// SIMATIC S7-200 SMART project (STEP 7-Micro/WIN SMART), CPU CR40

SYMBOL_TABLE 系统符号
Always_On        SM0.0    // 始终接通
First_Scan_On    SM0.1    // 仅在第一个扫描周期时接通
END_SYMBOL_TABLE

ORGANIZATION_BLOCK MAIN:OB1
TITLE=程序注释
BEGIN
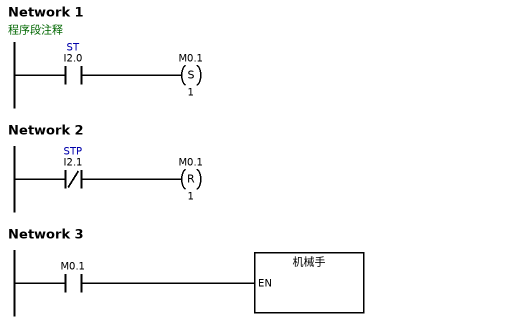
Network 1
// 程序段注释
LD     ST:I2.0
S      M0.1, 1
Network 2
LDN    STP:I2.1
R      M0.1, 1
Network 3
// (network saved uncompiled; LAD cells follow)
// row 0: c0 -| |- M0.1  c1 --  c2 [机械手 EN:=power@row0]
END_ORGANIZATION_BLOCK

SUBROUTINE_BLOCK 机械手:SBR0
TITLE=初始化，机械手复位
BEGIN
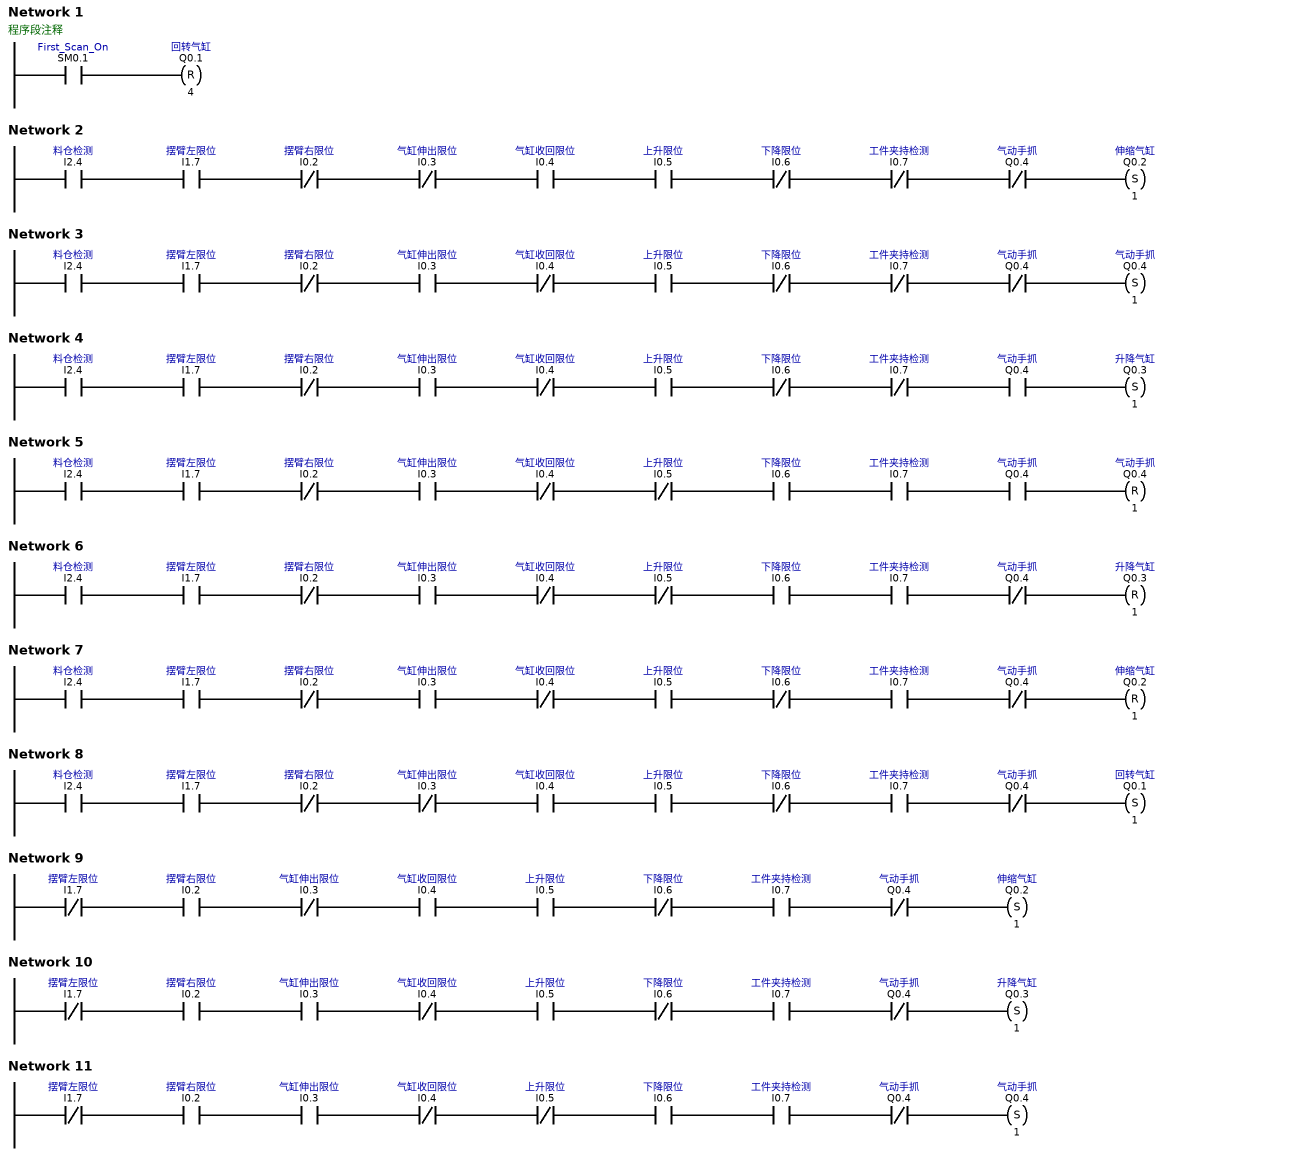
Network 1
// 程序段注释
LD     First_Scan_On:SM0.1
R      回转气缸:Q0.1, 4
Network 2
LD     料仓检测:I2.4
A      摆臂左限位:I1.7
AN     摆臂右限位:I0.2
AN     气缸伸出限位:I0.3
A      气缸收回限位:I0.4
A      上升限位:I0.5
AN     下降限位:I0.6
AN     工件夹持检测:I0.7
AN     气动手抓:Q0.4
S      伸缩气缸:Q0.2, 1
Network 3
LD     料仓检测:I2.4
A      摆臂左限位:I1.7
AN     摆臂右限位:I0.2
A      气缸伸出限位:I0.3
AN     气缸收回限位:I0.4
A      上升限位:I0.5
AN     下降限位:I0.6
AN     工件夹持检测:I0.7
AN     气动手抓:Q0.4
S      气动手抓:Q0.4, 1
Network 4
LD     料仓检测:I2.4
A      摆臂左限位:I1.7
AN     摆臂右限位:I0.2
A      气缸伸出限位:I0.3
AN     气缸收回限位:I0.4
A      上升限位:I0.5
AN     下降限位:I0.6
AN     工件夹持检测:I0.7
A      气动手抓:Q0.4
S      升降气缸:Q0.3, 1
Network 5
// 
// 
LD     料仓检测:I2.4
A      摆臂左限位:I1.7
AN     摆臂右限位:I0.2
A      气缸伸出限位:I0.3
AN     气缸收回限位:I0.4
AN     上升限位:I0.5
A      下降限位:I0.6
A      工件夹持检测:I0.7
A      气动手抓:Q0.4
R      气动手抓:Q0.4, 1
Network 6
// 
// 
LD     料仓检测:I2.4
A      摆臂左限位:I1.7
AN     摆臂右限位:I0.2
A      气缸伸出限位:I0.3
AN     气缸收回限位:I0.4
AN     上升限位:I0.5
A      下降限位:I0.6
A      工件夹持检测:I0.7
AN     气动手抓:Q0.4
R      升降气缸:Q0.3, 1
Network 7
// 
// 
LD     料仓检测:I2.4
A      摆臂左限位:I1.7
AN     摆臂右限位:I0.2
A      气缸伸出限位:I0.3
AN     气缸收回限位:I0.4
A      上升限位:I0.5
AN     下降限位:I0.6
A      工件夹持检测:I0.7
AN     气动手抓:Q0.4
R      伸缩气缸:Q0.2, 1
Network 8
// 
// 
LD     料仓检测:I2.4
A      摆臂左限位:I1.7
AN     摆臂右限位:I0.2
AN     气缸伸出限位:I0.3
A      气缸收回限位:I0.4
A      上升限位:I0.5
AN     下降限位:I0.6
A      工件夹持检测:I0.7
AN     气动手抓:Q0.4
S      回转气缸:Q0.1, 1
Network 9
// 
// 
// 
LDN    摆臂左限位:I1.7
A      摆臂右限位:I0.2
AN     气缸伸出限位:I0.3
A      气缸收回限位:I0.4
A      上升限位:I0.5
AN     下降限位:I0.6
A      工件夹持检测:I0.7
AN     气动手抓:Q0.4
S      伸缩气缸:Q0.2, 1
Network 10
// 
// 
// 
LDN    摆臂左限位:I1.7
A      摆臂右限位:I0.2
A      气缸伸出限位:I0.3
AN     气缸收回限位:I0.4
A      上升限位:I0.5
AN     下降限位:I0.6
A      工件夹持检测:I0.7
AN     气动手抓:Q0.4
S      升降气缸:Q0.3, 1
Network 11
// 
// 
// 
LDN    摆臂左限位:I1.7
A      摆臂右限位:I0.2
A      气缸伸出限位:I0.3
AN     气缸收回限位:I0.4
AN     上升限位:I0.5
A      下降限位:I0.6
A      工件夹持检测:I0.7
AN     气动手抓:Q0.4
S      气动手抓:Q0.4, 1
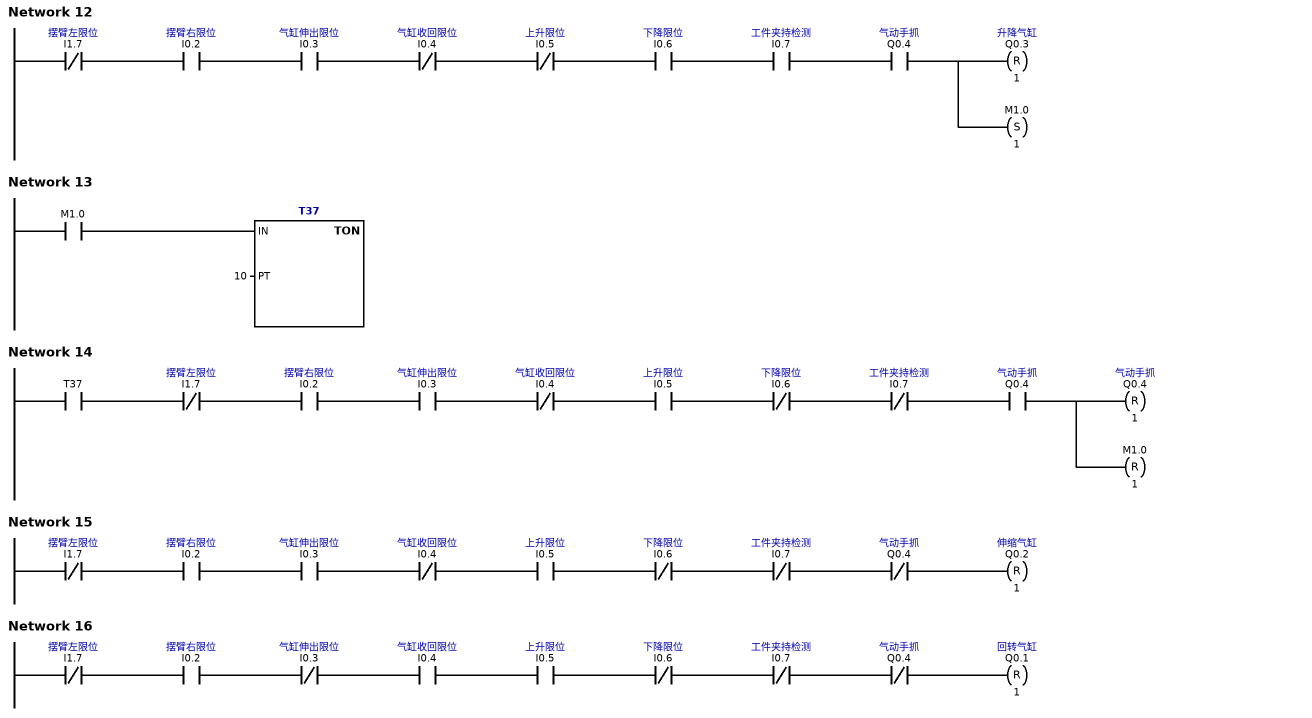
Network 12
// 
// 
// 
LDN    摆臂左限位:I1.7
A      摆臂右限位:I0.2
A      气缸伸出限位:I0.3
AN     气缸收回限位:I0.4
AN     上升限位:I0.5
A      下降限位:I0.6
A      工件夹持检测:I0.7
A      气动手抓:Q0.4
R      升降气缸:Q0.3, 1
S      M1.0, 1
Network 13
LD     M1.0
TON    T37, 10
Network 14
// 
// 
// 
LD     T37
AN     摆臂左限位:I1.7
A      摆臂右限位:I0.2
A      气缸伸出限位:I0.3
AN     气缸收回限位:I0.4
A      上升限位:I0.5
AN     下降限位:I0.6
AN     工件夹持检测:I0.7
A      气动手抓:Q0.4
R      气动手抓:Q0.4, 1
R      M1.0, 1
Network 15
// 
// 
// 
LDN    摆臂左限位:I1.7
A      摆臂右限位:I0.2
A      气缸伸出限位:I0.3
AN     气缸收回限位:I0.4
A      上升限位:I0.5
AN     下降限位:I0.6
AN     工件夹持检测:I0.7
AN     气动手抓:Q0.4
R      伸缩气缸:Q0.2, 1
Network 16
// 
// 
// 
LDN    摆臂左限位:I1.7
A      摆臂右限位:I0.2
AN     气缸伸出限位:I0.3
A      气缸收回限位:I0.4
A      上升限位:I0.5
AN     下降限位:I0.6
AN     工件夹持检测:I0.7
AN     气动手抓:Q0.4
R      回转气缸:Q0.1, 1
END_SUBROUTINE_BLOCK

SUBROUTINE_BLOCK 传送带:SBR1
TITLE=子程序注释
BEGIN
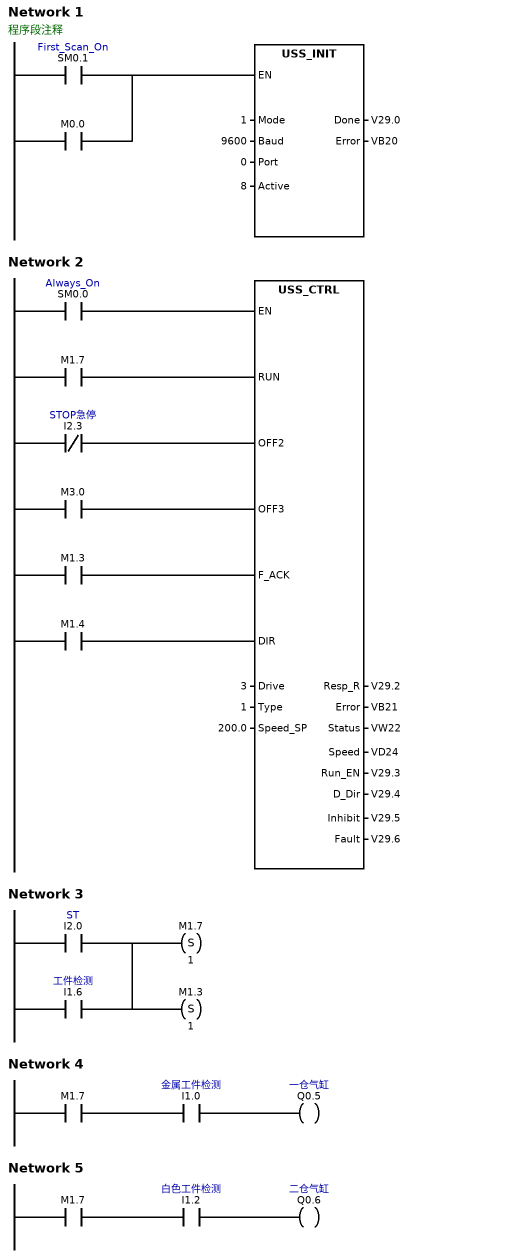
Network 1
// 程序段注释
LD     First_Scan_On:SM0.1
O      M0.0
CALL   USS_INIT:SBR3, 1, 9600, 0, 8, V29.0, VB20
Network 2
LD     Always_On:SM0.0
=      L60.0
LD     M1.7
=      L63.7
LDN    STOP急停:I2.3
=      L63.6
LD     M3.0
=      L63.5
LD     M1.3
=      L63.4
LD     M1.4
=      L63.3
LD     L60.0
CALL   USS_CTRL:SBR7, L63.7, L63.6, L63.5, L63.4, L63.3, 3, 1, 200.0, V29.2, VB21, VW22, VD24, V29.3, V29.4, V29.5, V29.6
Network 3
// (network saved uncompiled; LAD cells follow)
// row 0: c0 -| |- ST:I2.0 v  c1 -(S) M1.7, 1
// row 1: c0 -| |- 工件检测:I1.6 ^  c1 -(S) M1.3, 1
Network 4
LD     M1.7
A      金属工件检测:I1.0
=      一仓气缸:Q0.5
Network 5
LD     M1.7
A      白色工件检测:I1.2
=      二仓气缸:Q0.6
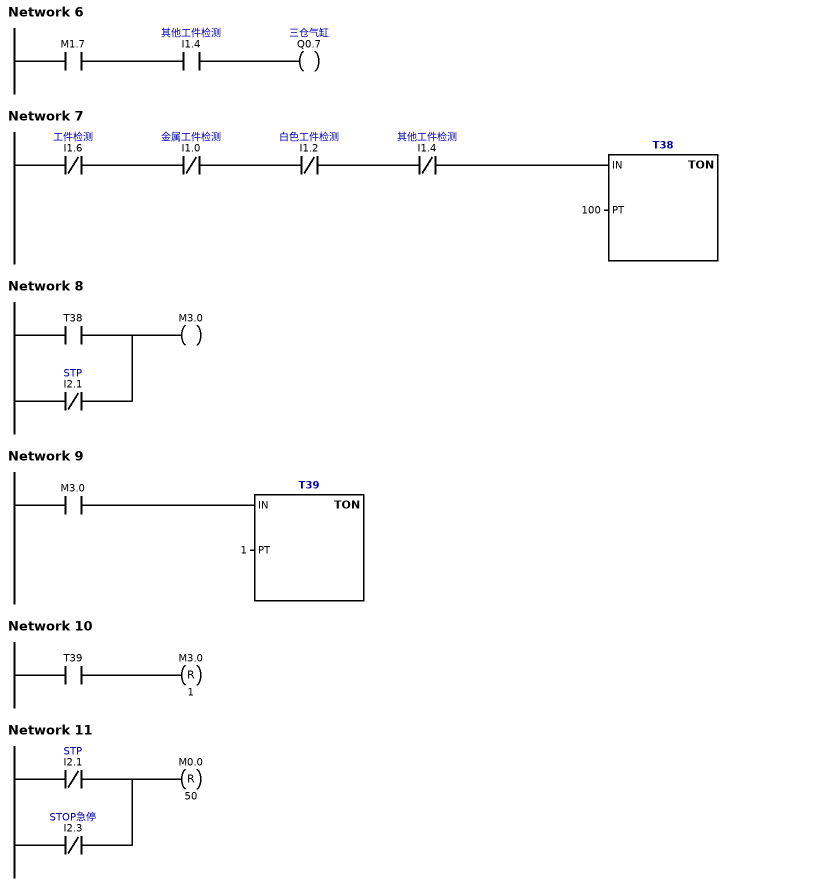
Network 6
LD     M1.7
A      其他工件检测:I1.4
=      三仓气缸:Q0.7
Network 7
LDN    工件检测:I1.6
AN     金属工件检测:I1.0
AN     白色工件检测:I1.2
AN     其他工件检测:I1.4
TON    T38, 100
Network 8
LD     T38
ON     STP:I2.1
=      M3.0
Network 9
LD     M3.0
TON    T39, 1
Network 10
LD     T39
R      M3.0, 1
Network 11
LDN    STP:I2.1
ON     STOP急停:I2.3
R      M0.0, 50
END_SUBROUTINE_BLOCK

// SBR3: protected block, not included

// SBR4: protected block, not included

// SBR5: protected block, not included

// SBR6: protected block, not included

// SBR7: protected block, not included

INTERRUPT_BLOCK 传送:INT0
TITLE=中断例程注释
BEGIN
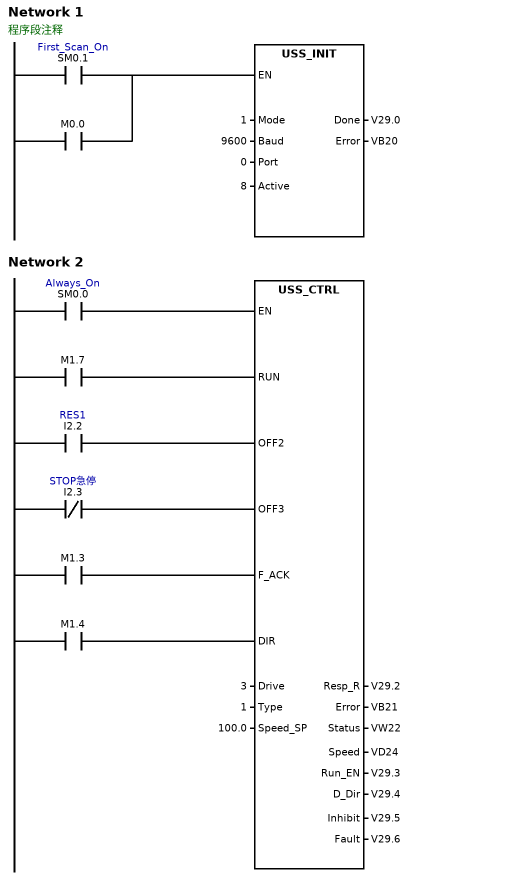
Network 1
// 程序段注释
LD     First_Scan_On:SM0.1
O      M0.0
CALL   USS_INIT:SBR3, 1, 9600, 0, 8, V29.0, VB20
Network 2
LD     Always_On:SM0.0
=      L60.0
LD     M1.7
=      L63.7
LD     RES1:I2.2
=      L63.6
LDN    STOP急停:I2.3
=      L63.5
LD     M1.3
=      L63.4
LD     M1.4
=      L63.3
LD     L60.0
CALL   USS_CTRL:SBR7, L63.7, L63.6, L63.5, L63.4, L63.3, 3, 1, 100.0, V29.2, VB21, VW22, VD24, V29.3, V29.4, V29.5, V29.6
END_INTERRUPT_BLOCK

// INT1: protected block, not included
